(* CoDeSys 2.3 export: ST_SENSOR_SWITCH.EXP *)

(* Data type *)
TYPE ST_SENSOR_SWITCH :
STRUCT
	Name : STRING;
	Desc : STRING;

	(*Alarm*)
	Alarm : ST_ALARM;

	Count  : REAL;


END_STRUCT
END_TYPE
